// TwinCAT 3 PLC project PLC_1
// ProgramVersion: 3.1.4024.0
// libraries:
//   Tc2_ModbusSrv, * (Beckhoff Automation GmbH)
//   Tc2_Standard, * (Beckhoff Automation GmbH)
//   Tc2_System, * (Beckhoff Automation GmbH)
//   Tc3_Module, * (Beckhoff Automation GmbH)
// project tree:
//   GVLs/ GVL.TcGVL
//   / PlcTask.TcTTO
//   POUs/ MAIN.TcPOU, ConveyorController.TcPOU
// real-time tasks:
//   TASK PlcTask: cycle T#10ms, priority 20, ADS port 350

CONFIGURATION PLC_1
    RESOURCE PLC ON TwinCAT3
        TASK PlcTask(INTERVAL := T#10ms, PRIORITY := 20);
        PROGRAM MAIN WITH PlcTask : MAIN;
    END_RESOURCE
END_CONFIGURATION

// ---- GVLs/GVL.TcGVL
{attribute 'qualified_only'}
VAR_GLOBAL
	mb_Input_Coils : ARRAY [0..5] OF BOOL;
	mb_Output_Coils : ARRAY [0..5] OF BOOL;
END_VAR

// ---- POUs/MAIN.TcPOU
PROGRAM MAIN
VAR
	Controller : ConveyorController;
END_VAR

Controller();

END_PROGRAM

// ---- POUs/ConveyorController.TcPOU
FUNCTION_BLOCK ConveyorController
VAR_INPUT
	ItemReady : BOOL;
	AtEntry : BOOL;
	AtExit : BOOL;
	FactoryIO_Run : BOOL;
END_VAR
VAR_OUTPUT
	EntryConveyor : BOOL;
	BufferConveyor : BOOL;
	Emitter : BOOL;
END_VAR
VAR
	ValueReached : BOOL;

	R_TRIG_0: R_TRIG;
	F_TRIG_0: F_TRIG;
	CTUD_0: CTUD;
	F_TRIG_1: F_TRIG;
	R_TRIG_1: R_TRIG;
	R_TRIG_2: R_TRIG;
	F_TRIG_2: F_TRIG;
END_VAR
VAR // added by the converter: edge detectors and wires of the graphical bodies
    _w1 : BOOL;
END_VAR

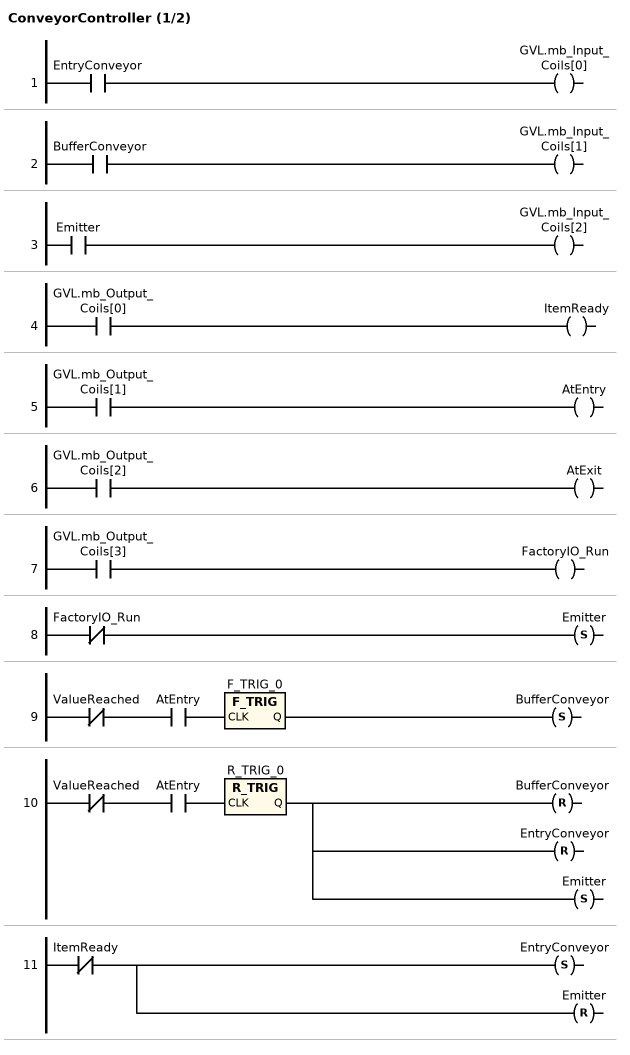
// NETWORK 1
GVL.mb_Input_Coils[0] := EntryConveyor;

// NETWORK 2
GVL.mb_Input_Coils[1] := BufferConveyor;

// NETWORK 3
GVL.mb_Input_Coils[2] := Emitter;

// NETWORK 4
ItemReady := GVL.mb_Output_Coils[0];

// NETWORK 5
AtEntry := GVL.mb_Output_Coils[1];

// NETWORK 6
AtExit := GVL.mb_Output_Coils[2];

// NETWORK 7
FactoryIO_Run := GVL.mb_Output_Coils[3];

// NETWORK 8
Emitter S= NOT FactoryIO_Run;

// NETWORK 9
F_TRIG_0(CLK := NOT ValueReached AND AtEntry); // F_TRIG
BufferConveyor S= F_TRIG_0.Q;

// NETWORK 10
R_TRIG_0(CLK := NOT ValueReached AND AtEntry); // R_TRIG
BufferConveyor R= R_TRIG_0.Q;
EntryConveyor R= R_TRIG_0.Q;
Emitter S= R_TRIG_0.Q;

// NETWORK 11
_w1 := NOT ItemReady;
EntryConveyor S= _w1;
Emitter R= _w1;

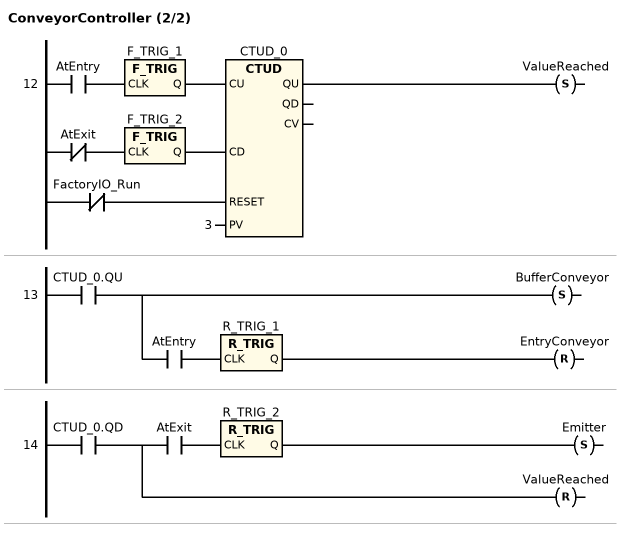
// NETWORK 12
F_TRIG_1(CLK := AtEntry); // F_TRIG
F_TRIG_2(CLK := NOT AtExit); // F_TRIG
CTUD_0(CU := F_TRIG_1.Q, CD := F_TRIG_2.Q, RESET := NOT FactoryIO_Run, PV := 3); // CTUD
ValueReached S= CTUD_0.QU;

// NETWORK 13
BufferConveyor S= CTUD_0.QU;
R_TRIG_1(CLK := CTUD_0.QU AND AtEntry); // R_TRIG
EntryConveyor R= R_TRIG_1.Q;

// NETWORK 14
R_TRIG_2(CLK := CTUD_0.QD AND AtExit); // R_TRIG
Emitter S= R_TRIG_2.Q;
ValueReached R= CTUD_0.QD;

END_FUNCTION_BLOCK
